// TIA Portal V17 export
// export: Created 2025-03-05T08:01:01.1286192Z, ExportSetting WithDefaults, DisplayName Totally Integrated Automation Portal, DisplayVersion V17 Update 8, DisplayName TIA Portal Openness, DisplayVersion V17 Update 8, DisplayName TIA Portal Version Control Interface, DisplayVersion V17, DisplayName SINAMICS Startdrive Advanced, DisplayVersion V17 SP2, DisplayName SINAMICS Startdrive G110M, G120, G120C, G120D, G120P, G115D, DisplayVersion V17 SP2, DisplayName SINAMICS Startdrive G130, G150, S120, S150, SINAMICS MV, S210, DisplayVersion V17 SP2, DisplayName STEP 7 Professional, DisplayVersion V17 Update 8, DisplayName SINUMERIK ONE STEP 7 Toolbox, DisplayVersion V17 Update 12, DisplayName SINUMERIK 840D sl STEP 7 Toolbox, DisplayVersion V17 Update 12, DisplayName STEP 7 Safety, DisplayVersion V17 Update 6, DisplayName WinCC Advanced, DisplayVersion V17 Update 8
DATA_BLOCK "LTLP_HMIProInterfaceData"   // DB501
{ S7_Optimized_Access := 'FALSE'; DB_Accessible_From_OPC_UA := 'FALSE' }
AUTHOR : TL_TYP6
FAMILY : TL
NAME : UDT_HMI
VERSION : 4.0
// stored: AutoNumber false, DBAccessibleFromOPCUA false, DBAccessibleFromWebserver true, InstanceOfName LTLP_typeHmiProInterface, InstanceOfType UDT, IsOnlyStoredInLoadMemory false, IsWriteProtectedInAS false
"LTLP_typeHmiProInterface"
   // VAR RETAIN
   //    nameStation : Array[1..8] of Char;
   //    noDBWorkpieceCount32 : Int;
   //    startDBWorkpieceCount32 : Int;
   //    cntWorkpiecetypes : Int;
   //    currentProtectLevel : Byte;
   //    eksIdent1 : Byte;
   //    eksIdent2 : Byte;
   //    eksIdent3 : Byte;
   //    eksIdent4 : Byte;
   //    eksIdent5 : Byte;
   //    eksIdent6 : Byte;
   //    eksIdent7 : Byte;
   //    eksOperatorIdentification : Byte;
   //    eksIdent8 : Byte;
   //    res24 : Array[24..31] of Byte;
   //    eksPLCSwitchover : Byte;
   //    res33 : Array[34..47] of Byte;
   //    byte480 : Byte;
   //    netIndex : Byte;
   //    resWinBDE : Array[50..53] of Byte;
   //    selWorkpiecetypePreselect : Word;
   //    selWorkpieceCountReset : Word;
   //    resetTotalCounter : Bool;
   //    resetDailyCounter : Bool;
   //    resetShiftCounter : Bool;
   //    res60 : Array[60..67] of Byte;
   //    codeWorkpiece : Word;
   //    selectProtectionDoors : Bool;
   //    reserve70p1 : Bool;
   //    reserve70p2 : Bool;
   //    reserve70p3 : Bool;
   //    reserve70p4 : Bool;
   //    reserve70p5 : Bool;
   //    reserve70p6 : Bool;
   //    reserve70p7 : Bool;
   //    reserve70p8 : Bool;
   //    reserve70p9 : Bool;
   //    reserve70p10 : Bool;
   //    reserve70p11 : Bool;
   //    reserve70p12 : Bool;
   //    reserve70p13 : Bool;
   //    reserve70p14 : Bool;
   //    reserve70p15 : Bool;
   //    noFunctionKeySubscreen : Word;
   //    selToolGroup : Byte;
   //    toolExtendingServiceLife : Bool;
   //    toolReactivating : Bool;
   //    toolDisable : Bool;
   //    res753 : Bool;
   //    res754 : Bool;
   //    res755 : Bool;
   //    res756 : Bool;
   //    res757 : Bool;
   //    controlPanelOk : Bool;
   //    pAutomaticMode : Bool;
   //    pSingleMode : Bool;
   //    pSingleStepMode : Bool;
   //    pSetupMode : Bool;
   //    pAllUnitsBack : Bool;
   //    pMachineOff : Bool;
   //    p6 : Bool;
   //    p7 : Bool;
   //    pPlus : Bool;
   //    pMinus : Bool;
   //    pEmergencyStop : Bool;
   //    pFaultWillBeCorrected : Bool;
   //    pStart : Bool;
   //    pBasicPosition : Bool;
   //    pMachineOn : Bool;
   //    pGroupAcknowledge : Bool;
   //    pReset : Bool;
   //    pLamptest : Bool;
   //    pRunmode_sweep : Bool;
   //    pMessageAcknowledge : Bool;
   //    pPartCounterReset : Bool;
   //    noFunctionLow : Byte;
   //    noFunctionHigh : Byte;
   //    pStopAfterEndOfCycle : Bool;
   //    pImmediateStop : Bool;
   //    pBridgeEnablingButton : Bool;
   //    pConnectEnablingButton : Bool;
   //    pLockReleaseProtectDoors : Bool;
   //    pMediaOn : Bool;
   //    pMediaOff : Bool;
   //    noSoftKey : Byte;
   //    noFunctionKey : Byte;
   //    noScreenId : Word;
   //    automaticModeCompleteMachine : Bool;
   //    automaticMode : Bool;
   //    singleMode : Bool;
   //    singleStepMode : Bool;
   //    setupMode : Bool;
   //    completionReport : Bool;
   //    gotoBasicPosition : Bool;
   //    reachedBasicPosition : Bool;
   //    startJog : Bool;
   //    immediateStop : Bool;
   //    selStopAfterEndOfCycle : Bool;
   //    reachedStopAfterEndOfCycle : Bool;
   //    motionPlus : Bool;
   //    motionMinus : Bool;
   //    machineUnitOn : Bool;
   //    machineUnitOff : Bool;
   //    allUnitsBack : Bool;
   //    accessAuthorized : Bool;
   //    generalFault : Bool;
   //    executionFault : Bool;
   //    warningOperationalMessage : Bool;
   //    completeMachineFault : Bool;
   //    completeMachineBasicPosition : Bool;
   //    completeMachineCompletReport { ExternalWritable := 'False'} : Bool;
   //    faPartMachining : Bool;
   //    load : Bool;
   //    withoutMachining : Bool;
   //    toolGroupAckOrEnable : Bool;
   //    readyAutomaticStart : Bool;
   //    res895 : Bool;
   //    res896 : Bool;
   //    res897 : Bool;
   //    cycletypes : Array[1..16] of Bool;
   //    protectiveDoorBridged : Bool;
   //    faultWillBeCorrected : Bool;
   //    BridgeEnablingButton : Bool;
   //    connectEnablingButton : Bool;
   //    groupBitProtectDoorsopen : Bool;
   //    headerSwitchover : Bool;
   //    machineUtilization : Bool;
   //    message : Bool;
   //    logisticsFault : Bool;
   //    globalSupplyOutfeed : Bool;
   //    idleCycles : Bool;
   //    toolChangeAlarm : Bool;
   //    automaticToolChangePosition : Bool;
   //    updateRequest : Bool;
   //    toolChangeWarning : Bool;
   //    learnToolChangeSystemActive : Bool;
   //    headerText1 : Bool;
   //    headerText2 : Bool;
   //    headerText3 : Bool;
   //    headerText4 : Bool;
   //    headerText5 : Bool;
   //    headerText6 : Bool;
   //    headerText7 : Bool;
   //    headerText8 : Bool;
   //    automaticStart : Bool;
   //    manualMode : Bool;
   //    transportPosition : Bool;
   //    handHeldUnit : Bool;
   //    mediaOn : Bool;
   //    mediaOff : Bool;
   //    lockReleaseProtectDoors : Bool;
   //    lockingScreenSwitchover : Bool;
   //    exitIsOccupied : Bool;
   //    noPartAtInfeed : Bool;
   //    noFeedParts : Bool;
   //    changeLanguage : Bool;
   //    TriggBitReadPartId : Bool;
   //    cycleBitShiftRegPartId : Bool;
   //    disableDataAvailable : Bool;
   //    upsResponded : Bool;
   //    pageId : Byte;
   //    shiftNumber : Byte;
   //    partsPerCycle : Byte;
   //    taskTriggFeedbackRecipe : Byte;
   //    noControlRecipe : Byte;
   //    nameScreenRecipe : Array[1..27] of Char;
   //    movement1EndPosLeft : Bool;   // Setup screen: left end position of movement reached
   //    movement1EndPosRight : Bool;   // Setup screen: right end position of movement reached
   //    movement2EndPosLeft : Bool;   // Setup screen: left end position of movement reached
   //    movement2EndPosRight : Bool;   // Setup screen: right end position of movement reached
   //    movement3EndPosLeft : Bool;   // Setup screen: left end position of movement reached
   //    movement3EndPosRight : Bool;   // Setup screen: right end position of movement reached
   //    movement4EndPosLeft : Bool;   // Setup screen: left end position of movement reached
   //    movement4EndPosRight : Bool;   // Setup screen: right end position of movement reached
   //    movement5EndPosLeft : Bool;   // Setup screen: left end position of movement reached
   //    movement5EndPosRight : Bool;   // Setup screen: right end position of movement reached
   //    movement6EndPosLeft : Bool;   // Setup screen: left end position of movement reached
   //    movement6EndPosRight : Bool;   // Setup screen: right end position of movement reached
   //    movement7EndPosLeft : Bool;   // Setup screen: left end position of movement reached
   //    movement7EndPosRight : Bool;   // Setup screen: right end position of movement reached
   //    movement8EndPosLeft : Bool;   // Setup screen: left end position of movement reached
   //    movement8EndPosRight : Bool;   // Setup screen: right end position of movement reached
   //    movement9EndPosLeft : Bool;   // Setup screen: left end position of movement reached
   //    movement9EndPosRight : Bool;   // Setup screen: right end position of movement reached
   //    movement10EndPosLeft : Bool;   // Setup screen: left end position of movement reached
   //    movement10EndPosRight : Bool;   // Setup screen: right end position of movement reached
   //    movement11EndPosLeft : Bool;   // Setup screen: left end position of movement reached
   //    movement11EndPosRight : Bool;   // Setup screen: right end position of movement reached
   //    movement12EndPosLeft : Bool;   // Setup screen: left end position of movement reached
   //    movement12EndPosRight : Bool;   // Setup screen: right end position of movement reached
   //    movement13EndPosLeft : Bool;   // Setup screen: left end position of movement reached
   //    movement13EndPosRight : Bool;   // Setup screen: right end position of movement reached
   //    movement14EndPosLeft : Bool;   // Setup screen: left end position of movement reached
   //    movement14EndPosRight : Bool;   // Setup screen: right end position of movement reached
   //    movement15EndPosLeft : Bool;   // Setup screen: left end position of movement reached
   //    movement15EndPosRight : Bool;   // Setup screen: right end position of movement reached
   //    movement16EndPosLeft : Bool;   // Setup screen: left end position of movement reached
   //    movement16EndPosRight : Bool;   // Setup screen: right end position of movement reached
   //    movement17EndPosLeft : Bool;   // Setup screen: left end position of movement reached
   //    movement17EndPosRight : Bool;   // Setup screen: right end position of movement reached
   //    movement18EndPosLeft : Bool;   // Setup screen: left end position of movement reached
   //    movement18EndPosRight : Bool;   // Setup screen: right end position of movement reached
   //    movement19EndPosLeft : Bool;   // Setup screen: left end position of movement reached
   //    movement19EndPosRight : Bool;   // Setup screen: right end position of movement reached
   //    movement20EndPosLeft : Bool;   // Setup screen: left end position of movement reached
   //    movement20EndPosRight : Bool;   // Setup screen: right end position of movement reached
   //    movement21EndPosLeft : Bool;   // Setup screen: left end position of movement reached
   //    movement21EndPosRight : Bool;   // Setup screen: right end position of movement reached
   //    movement22EndPosLeft : Bool;   // Setup screen: left end position of movement reached
   //    movement22EndPosRight : Bool;   // Setup screen: right end position of movement reached
   //    movement23EndPosLeft : Bool;   // Setup screen: left end position of movement reached
   //    movement23EndPosRight : Bool;   // Setup screen: right end position of movement reached
   //    movement24EndPosLeft : Bool;   // Setup screen: left end position of movement reached
   //    movement24EndPosRight : Bool;   // Setup screen: right end position of movement reached
   //    movement25EndPosLeft : Bool;   // Setup screen: left end position of movement reached
   //    movement25EndPosRight : Bool;   // Setup screen: right end position of movement reached
   //    movement26EndPosLeft : Bool;   // Setup screen: left end position of movement reached
   //    movement26EndPosRight : Bool;   // Setup screen: right end position of movement reached
   //    movement27EndPosLeft : Bool;   // Setup screen: left end position of movement reached
   //    movement27EndPosRight : Bool;   // Setup screen: right end position of movement reached
   //    movement28EndPosLeft : Bool;   // Setup screen: left end position of movement reached
   //    movement28EndPosRight : Bool;   // Setup screen: right end position of movement reached
   //    movement29EndPosLeft : Bool;   // Setup screen: left end position of movement reached
   //    movement29EndPosRight : Bool;   // Setup screen: right end position of movement reached
   //    movement30EndPosLeft : Bool;   // Setup screen: left end position of movement reached
   //    movement30EndPosRight : Bool;   // Setup screen: right end position of movement reached
   //    movement31EndPosLeft : Bool;   // Setup screen: left end position of movement reached
   //    movement31EndPosRight : Bool;   // Setup screen: right end position of movement reached
   //    movement32EndPosLeft : Bool;   // Setup screen: left end position of movement reached
   //    movement32EndPosRight : Bool;   // Setup screen: right end position of movement reached
   //    movement33EndPosLeft : Bool;   // Setup screen: left end position of movement reached
   //    movement33EndPosRight : Bool;   // Setup screen: right end position of movement reached
   //    movement34EndPosLeft : Bool;   // Setup screen: left end position of movement reached
   //    movement34EndPosRight : Bool;   // Setup screen: right end position of movement reached
   //    movement35EndPosLeft : Bool;   // Setup screen: left end position of movement reached
   //    movement35EndPosRight : Bool;   // Setup screen: right end position of movement reached
   //    movement36EndPosLeft : Bool;   // Setup screen: left end position of movement reached
   //    movement36EndPosRight : Bool;   // Setup screen: right end position of movement reached
   //    movement37EndPosLeft : Bool;   // Setup screen: left end position of movement reached
   //    movement37EndPosRight : Bool;   // Setup screen: right end position of movement reached
   //    movement38EndPosLeft : Bool;   // Setup screen: left end position of movement reached
   //    movement38EndPosRight : Bool;   // Setup screen: right end position of movement reached
   //    movement39EndPosLeft : Bool;   // Setup screen: left end position of movement reached
   //    movement39EndPosRight : Bool;   // Setup screen: right end position of movement reached
   //    movement40EndPosLeft : Bool;   // Setup screen: left end position of movement reached
   //    movement40EndPosRight : Bool;   // Setup screen: right end position of movement reached
   //    movement41EndPosLeft : Bool;   // Setup screen: left end position of movement reached
   //    movement41EndPosRight : Bool;   // Setup screen: right end position of movement reached
   //    movement42EndPosLeft : Bool;   // Setup screen: left end position of movement reached
   //    movement42EndPosRight : Bool;   // Setup screen: right end position of movement reached
   //    movement43EndPosLeft : Bool;   // Setup screen: left end position of movement reached
   //    movement43EndPosRight : Bool;   // Setup screen: right end position of movement reached
   //    movement44EndPosLeft : Bool;   // Setup screen: left end position of movement reached
   //    movement44EndPosRight : Bool;   // Setup screen: right end position of movement reached
   //    movement45EndPosLeft : Bool;   // Setup screen: left end position of movement reached
   //    movement45EndPosRight : Bool;   // Setup screen: right end position of movement reached
   //    movement46EndPosLeft : Bool;   // Setup screen: left end position of movement reached
   //    movement46EndPosRight : Bool;   // Setup screen: right end position of movement reached
   //    movement47EndPosLeft : Bool;   // Setup screen: left end position of movement reached
   //    movement47EndPosRight : Bool;   // Setup screen: right end position of movement reached
   //    movement48EndPosLeft : Bool;   // Setup screen: left end position of movement reached
   //    movement48EndPosRight : Bool;   // Setup screen: right end position of movement reached
   //    movement49EndPosLeft : Bool;   // Setup screen: left end position of movement reached
   //    movement49EndPosRight : Bool;   // Setup screen: right end position of movement reached
   //    movement50EndPosLeft : Bool;   // Setup screen: left end position of movement reached
   //    movement50EndPosRight : Bool;   // Setup screen: right end position of movement reached
   //    movement51EndPosLeft : Bool;   // Setup screen: left end position of movement reached
   //    movement51EndPosRight : Bool;   // Setup screen: right end position of movement reached
   //    movement52EndPosLeft : Bool;   // Setup screen: left end position of movement reached
   //    movement52EndPosRight : Bool;   // Setup screen: right end position of movement reached
   //    movement53EndPosLeft : Bool;   // Setup screen: left end position of movement reached
   //    movement53EndPosRight : Bool;   // Setup screen: right end position of movement reached
   //    movement54EndPosLeft : Bool;   // Setup screen: left end position of movement reached
   //    movement54EndPosRight : Bool;   // Setup screen: right end position of movement reached
   //    movement55EndPosLeft : Bool;   // Setup screen: left end position of movement reached
   //    movement55EndPosRight : Bool;   // Setup screen: right end position of movement reached
   //    movement56EndPosLeft : Bool;   // Setup screen: left end position of movement reached
   //    movement56EndPosRight : Bool;   // Setup screen: right end position of movement reached
   //    movement57EndPosLeft : Bool;   // Setup screen: left end position of movement reached
   //    movement57EndPosRight : Bool;   // Setup screen: right end position of movement reached
   //    movement58EndPosLeft : Bool;   // Setup screen: left end position of movement reached
   //    movement58EndPosRight : Bool;   // Setup screen: right end position of movement reached
   //    movement59EndPosLeft : Bool;   // Setup screen: left end position of movement reached
   //    movement59EndPosRight : Bool;   // Setup screen: right end position of movement reached
   //    movement60EndPosLeft : Bool;   // Setup screen: left end position of movement reached
   //    movement60EndPosRight : Bool;   // Setup screen: right end position of movement reached
   //    movement61EndPosLeft : Bool;   // Setup screen: left end position of movement reached
   //    movement61EndPosRight : Bool;   // Setup screen: right end position of movement reached
   //    movement62EndPosLeft : Bool;   // Setup screen: left end position of movement reached
   //    movement62EndPosRight : Bool;   // Setup screen: right end position of movement reached
   //    movement63EndPosLeft : Bool;   // Setup screen: left end position of movement reached
   //    movement63EndPosRight : Bool;   // Setup screen: right end position of movement reached
   //    movement64EndPosLeft : Bool;   // Setup screen: left end position of movement reached
   //    movement64EndPosRight : Bool;   // Setup screen: right end position of movement reached
   //    movement65EndPosLeft : Bool;   // Setup screen: left end position of movement reached
   //    movement65EndPosRight : Bool;   // Setup screen: right end position of movement reached
   //    movement66EndPosLeft : Bool;   // Setup screen: left end position of movement reached
   //    movement66EndPosRight : Bool;   // Setup screen: right end position of movement reached
   //    movement67EndPosLeft : Bool;   // Setup screen: left end position of movement reached
   //    movement67EndPosRight : Bool;   // Setup screen: right end position of movement reached
   //    movement68EndPosLeft : Bool;   // Setup screen: left end position of movement reached
   //    movement68EndPosRight : Bool;   // Setup screen: right end position of movement reached
   //    movement69EndPosLeft : Bool;   // Setup screen: left end position of movement reached
   //    movement69EndPosRight : Bool;   // Setup screen: right end position of movement reached
   //    movement70EndPosLeft : Bool;   // Setup screen: left end position of movement reached
   //    movement70EndPosRight : Bool;   // Setup screen: right end position of movement reached
   //    movement71EndPosLeft : Bool;   // Setup screen: left end position of movement reached
   //    movement71EndPosRight : Bool;   // Setup screen: right end position of movement reached
   //    movement72EndPosLeft : Bool;   // Setup screen: left end position of movement reached
   //    movement72EndPosRight : Bool;   // Setup screen: right end position of movement reached
   //    movement73EndPosLeft : Bool;   // Setup screen: left end position of movement reached
   //    movement73EndPosRight : Bool;   // Setup screen: right end position of movement reached
   //    movement74EndPosLeft : Bool;   // Setup screen: left end position of movement reached
   //    movement74EndPosRight : Bool;   // Setup screen: right end position of movement reached
   //    movement75EndPosLeft : Bool;   // Setup screen: left end position of movement reached
   //    movement75EndPosRight : Bool;   // Setup screen: right end position of movement reached
   //    movement76EndPosLeft : Bool;   // Setup screen: left end position of movement reached
   //    movement76EndPosRight : Bool;   // Setup screen: right end position of movement reached
   //    movement77EndPosLeft : Bool;   // Setup screen: left end position of movement reached
   //    movement77EndPosRight : Bool;   // Setup screen: right end position of movement reached
   //    movement78EndPosLeft : Bool;   // Setup screen: left end position of movement reached
   //    movement78EndPosRight : Bool;   // Setup screen: right end position of movement reached
   //    movement79EndPosLeft : Bool;   // Setup screen: left end position of movement reached
   //    movement79EndPosRight : Bool;   // Setup screen: right end position of movement reached
   //    movement80EndPosLeft : Bool;   // Setup screen: left end position of movement reached
   //    movement80EndPosRight : Bool;   // Setup screen: right end position of movement reached
   //    movement81EndPosLeft : Bool;   // Setup screen: left end position of movement reached
   //    movement81EndPosRight : Bool;   // Setup screen: right end position of movement reached
   //    movement82EndPosLeft : Bool;   // Setup screen: left end position of movement reached
   //    movement82EndPosRight : Bool;   // Setup screen: right end position of movement reached
   //    movement83EndPosLeft : Bool;   // Setup screen: left end position of movement reached
   //    movement83EndPosRight : Bool;   // Setup screen: right end position of movement reached
   //    movement84EndPosLeft : Bool;   // Setup screen: left end position of movement reached
   //    movement84EndPosRight : Bool;   // Setup screen: right end position of movement reached
   //    movement85EndPosLeft : Bool;   // Setup screen: left end position of movement reached
   //    movement85EndPosRight : Bool;   // Setup screen: right end position of movement reached
   //    movement86EndPosLeft : Bool;   // Setup screen: left end position of movement reached
   //    movement86EndPosRight : Bool;   // Setup screen: right end position of movement reached
   //    movement87EndPosLeft : Bool;   // Setup screen: left end position of movement reached
   //    movement87EndPosRight : Bool;   // Setup screen: right end position of movement reached
   //    movement88EndPosLeft : Bool;   // Setup screen: left end position of movement reached
   //    movement88EndPosRight : Bool;   // Setup screen: right end position of movement reached
   //    movement89EndPosLeft : Bool;   // Setup screen: left end position of movement reached
   //    movement89EndPosRight : Bool;   // Setup screen: right end position of movement reached
   //    movement90EndPosLeft : Bool;   // Setup screen: left end position of movement reached
   //    movement90EndPosRight : Bool;   // Setup screen: right end position of movement reached
   //    movement91EndPosLeft : Bool;   // Setup screen: left end position of movement reached
   //    movement91EndPosRight : Bool;   // Setup screen: right end position of movement reached
   //    movement92EndPosLeft : Bool;   // Setup screen: left end position of movement reached
   //    movement92EndPosRight : Bool;   // Setup screen: right end position of movement reached
   //    movement93EndPosLeft : Bool;   // Setup screen: left end position of movement reached
   //    movement93EndPosRight : Bool;   // Setup screen: right end position of movement reached
   //    movement94EndPosLeft : Bool;   // Setup screen: left end position of movement reached
   //    movement94EndPosRight : Bool;   // Setup screen: right end position of movement reached
   //    movement95EndPosLeft : Bool;   // Setup screen: left end position of movement reached
   //    movement95EndPosRight : Bool;   // Setup screen: right end position of movement reached
   //    movement96EndPosLeft : Bool;   // Setup screen: left end position of movement reached
   //    movement96EndPosRight : Bool;   // Setup screen: right end position of movement reached
   //    movement97EndPosLeft : Bool;   // Setup screen: left end position of movement reached
   //    movement97EndPosRight : Bool;   // Setup screen: right end position of movement reached
   //    movement98EndPosLeft : Bool;   // Setup screen: left end position of movement reached
   //    movement98EndPosRight : Bool;   // Setup screen: right end position of movement reached
   //    movement99EndPosLeft : Bool;   // Setup screen: left end position of movement reached
   //    movement99EndPosRight : Bool;   // Setup screen: right end position of movement reached
   //    movement100EndPosLeft : Bool;   // Setup screen: left end position of movement reached
   //    movement100EndPosRight : Bool;   // Setup screen: right end position of movement reached
   //    movement101EndPosLeft : Bool;   // Setup screen: left end position of movement reached
   //    movement101EndPosRight : Bool;   // Setup screen: right end position of movement reached
   //    movement102EndPosLeft : Bool;   // Setup screen: left end position of movement reached
   //    movement102EndPosRight : Bool;   // Setup screen: right end position of movement reached
   //    movement103EndPosLeft : Bool;   // Setup screen: left end position of movement reached
   //    movement103EndPosRight : Bool;   // Setup screen: right end position of movement reached
   //    movement104EndPosLeft : Bool;   // Setup screen: left end position of movement reached
   //    movement104EndPosRight : Bool;   // Setup screen: right end position of movement reached
   //    movement105EndPosLeft : Bool;   // Setup screen: left end position of movement reached
   //    movement105EndPosRight : Bool;   // Setup screen: right end position of movement reached
   //    movement106EndPosLeft : Bool;   // Setup screen: left end position of movement reached
   //    movement106EndPosRight : Bool;   // Setup screen: right end position of movement reached
   //    movement107EndPosLeft : Bool;   // Setup screen: left end position of movement reached
   //    movement107EndPosRight : Bool;   // Setup screen: right end position of movement reached
   //    movement108EndPosLeft : Bool;   // Setup screen: left end position of movement reached
   //    movement108EndPosRight : Bool;   // Setup screen: right end position of movement reached
   //    movement109EndPosLeft : Bool;   // Setup screen: left end position of movement reached
   //    movement109EndPosRight : Bool;   // Setup screen: right end position of movement reached
   //    movement110EndPosLeft : Bool;   // Setup screen: left end position of movement reached
   //    movement110EndPosRight : Bool;   // Setup screen: right end position of movement reached
   //    movement111EndPosLeft : Bool;   // Setup screen: left end position of movement reached
   //    movement111EndPosRight : Bool;   // Setup screen: right end position of movement reached
   //    movement112EndPosLeft : Bool;   // Setup screen: left end position of movement reached
   //    movement112EndPosRight : Bool;   // Setup screen: right end position of movement reached
   //    movement113EndPosLeft : Bool;   // Setup screen: left end position of movement reached
   //    movement113EndPosRight : Bool;   // Setup screen: right end position of movement reached
   //    movement114EndPosLeft : Bool;   // Setup screen: left end position of movement reached
   //    movement114EndPosRight : Bool;   // Setup screen: right end position of movement reached
   //    movement115EndPosLeft : Bool;   // Setup screen: left end position of movement reached
   //    movement115EndPosRight : Bool;   // Setup screen: right end position of movement reached
   //    movement116EndPosLeft : Bool;   // Setup screen: left end position of movement reached
   //    movement116EndPosRight : Bool;   // Setup screen: right end position of movement reached
   //    movement117EndPosLeft : Bool;   // Setup screen: left end position of movement reached
   //    movement117EndPosRight : Bool;   // Setup screen: right end position of movement reached
   //    movement118EndPosLeft : Bool;   // Setup screen: left end position of movement reached
   //    movement118EndPosRight : Bool;   // Setup screen: right end position of movement reached
   //    movement119EndPosLeft : Bool;   // Setup screen: left end position of movement reached
   //    movement119EndPosRight : Bool;   // Setup screen: right end position of movement reached
   //    movement120EndPosLeft : Bool;   // Setup screen: left end position of movement reached
   //    movement120EndPosRight : Bool;   // Setup screen: right end position of movement reached
   //    movement121EndPosLeft : Bool;   // Setup screen: left end position of movement reached
   //    movement121EndPosRight : Bool;   // Setup screen: right end position of movement reached
   //    movement122EndPosLeft : Bool;   // Setup screen: left end position of movement reached
   //    movement122EndPosRight : Bool;   // Setup screen: right end position of movement reached
   //    movement123EndPosLeft : Bool;   // Setup screen: left end position of movement reached
   //    movement123EndPosRight : Bool;   // Setup screen: right end position of movement reached
   //    movement124EndPosLeft : Bool;   // Setup screen: left end position of movement reached
   //    movement124EndPosRight : Bool;   // Setup screen: right end position of movement reached
   //    movement125EndPosLeft : Bool;   // Setup screen: left end position of movement reached
   //    movement125EndPosRight : Bool;   // Setup screen: right end position of movement reached
   //    movement126EndPosLeft : Bool;   // Setup screen: left end position of movement reached
   //    movement126EndPosRight : Bool;   // Setup screen: right end position of movement reached
   //    movement127EndPosLeft : Bool;   // Setup screen: left end position of movement reached
   //    movement127EndPosRight : Bool;   // Setup screen: right end position of movement reached
   //    movement128EndPosLeft : Bool;   // Setup screen: left end position of movement reached
   //    movement128EndPosRight : Bool;   // Setup screen: right end position of movement reached
   //    movement129EndPosLeft : Bool;   // Setup screen: left end position of movement reached
   //    movement129EndPosRight : Bool;   // Setup screen: right end position of movement reached
   //    movement130EndPosLeft : Bool;   // Setup screen: left end position of movement reached
   //    movement130EndPosRight : Bool;   // Setup screen: right end position of movement reached
   //    movement131EndPosLeft : Bool;   // Setup screen: left end position of movement reached
   //    movement131EndPosRight : Bool;   // Setup screen: right end position of movement reached
   //    movement132EndPosLeft : Bool;   // Setup screen: left end position of movement reached
   //    movement132EndPosRight : Bool;   // Setup screen: right end position of movement reached
   //    movement133EndPosLeft : Bool;   // Setup screen: left end position of movement reached
   //    movement133EndPosRight : Bool;   // Setup screen: right end position of movement reached
   //    movement134EndPosLeft : Bool;   // Setup screen: left end position of movement reached
   //    movement134EndPosRight : Bool;   // Setup screen: right end position of movement reached
   //    movement135EndPosLeft : Bool;   // Setup screen: left end position of movement reached
   //    movement135EndPosRight : Bool;   // Setup screen: right end position of movement reached
   //    movement136EndPosLeft : Bool;   // Setup screen: left end position of movement reached
   //    movement136EndPosRight : Bool;   // Setup screen: right end position of movement reached
   //    movement137EndPosLeft : Bool;   // Setup screen: left end position of movement reached
   //    movement137EndPosRight : Bool;   // Setup screen: right end position of movement reached
   //    movement138EndPosLeft : Bool;   // Setup screen: left end position of movement reached
   //    movement138EndPosRight : Bool;   // Setup screen: right end position of movement reached
   //    movement139EndPosLeft : Bool;   // Setup screen: left end position of movement reached
   //    movement139EndPosRight : Bool;   // Setup screen: right end position of movement reached
   //    movement140EndPosLeft : Bool;   // Setup screen: left end position of movement reached
   //    movement140EndPosRight : Bool;   // Setup screen: right end position of movement reached
   //    movement141EndPosLeft : Bool;   // Setup screen: left end position of movement reached
   //    movement141EndPosRight : Bool;   // Setup screen: right end position of movement reached
   //    movement142EndPosLeft : Bool;   // Setup screen: left end position of movement reached
   //    movement142EndPosRight : Bool;   // Setup screen: right end position of movement reached
   //    movement143EndPosLeft : Bool;   // Setup screen: left end position of movement reached
   //    movement143EndPosRight : Bool;   // Setup screen: right end position of movement reached
   //    movement144EndPosLeft : Bool;   // Setup screen: left end position of movement reached
   //    movement144EndPosRight : Bool;   // Setup screen: right end position of movement reached
   //    movement145EndPosLeft : Bool;   // Setup screen: left end position of movement reached
   //    movement145EndPosRight : Bool;   // Setup screen: right end position of movement reached
   //    movement146EndPosLeft : Bool;   // Setup screen: left end position of movement reached
   //    movement146EndPosRight : Bool;   // Setup screen: right end position of movement reached
   //    movement147EndPosLeft : Bool;   // Setup screen: left end position of movement reached
   //    movement147EndPosRight : Bool;   // Setup screen: right end position of movement reached
   //    movement148EndPosLeft : Bool;   // Setup screen: left end position of movement reached
   //    movement148EndPosRight : Bool;   // Setup screen: right end position of movement reached
   //    movement149EndPosLeft : Bool;   // Setup screen: left end position of movement reached
   //    movement149EndPosRight : Bool;   // Setup screen: right end position of movement reached
   //    movement150EndPosLeft : Bool;   // Setup screen: left end position of movement reached
   //    movement150EndPosRight : Bool;   // Setup screen: right end position of movement reached
   //    movement151EndPosLeft : Bool;   // Setup screen: left end position of movement reached
   //    movement151EndPosRight : Bool;   // Setup screen: right end position of movement reached
   //    movement152EndPosLeft : Bool;   // Setup screen: left end position of movement reached
   //    movement152EndPosRight : Bool;   // Setup screen: right end position of movement reached
   //    movement153EndPosLeft : Bool;   // Setup screen: left end position of movement reached
   //    movement153EndPosRight : Bool;   // Setup screen: right end position of movement reached
   //    movement154EndPosLeft : Bool;   // Setup screen: left end position of movement reached
   //    movement154EndPosRight : Bool;   // Setup screen: right end position of movement reached
   //    movement155EndPosLeft : Bool;   // Setup screen: left end position of movement reached
   //    movement155EndPosRight : Bool;   // Setup screen: right end position of movement reached
   //    movement156EndPosLeft : Bool;   // Setup screen: left end position of movement reached
   //    movement156EndPosRight : Bool;   // Setup screen: right end position of movement reached
   //    movement157EndPosLeft : Bool;   // Setup screen: left end position of movement reached
   //    movement157EndPosRight : Bool;   // Setup screen: right end position of movement reached
   //    movement158EndPosLeft : Bool;   // Setup screen: left end position of movement reached
   //    movement158EndPosRight : Bool;   // Setup screen: right end position of movement reached
   //    movement159EndPosLeft : Bool;   // Setup screen: left end position of movement reached
   //    movement159EndPosRight : Bool;   // Setup screen: right end position of movement reached
   //    movement160EndPosLeft : Bool;   // Setup screen: left end position of movement reached
   //    movement160EndPosRight : Bool;   // Setup screen: right end position of movement reached
   //    movement161EndPosLeft : Bool;   // Setup screen: left end position of movement reached
   //    movement161EndPosRight : Bool;   // Setup screen: right end position of movement reached
   //    movement162EndPosLeft : Bool;   // Setup screen: left end position of movement reached
   //    movement162EndPosRight : Bool;   // Setup screen: right end position of movement reached
   //    movement163EndPosLeft : Bool;   // Setup screen: left end position of movement reached
   //    movement163EndPosRight : Bool;   // Setup screen: right end position of movement reached
   //    movement164EndPosLeft : Bool;   // Setup screen: left end position of movement reached
   //    movement164EndPosRight : Bool;   // Setup screen: right end position of movement reached
   //    movement165EndPosLeft : Bool;   // Setup screen: left end position of movement reached
   //    movement165EndPosRight : Bool;   // Setup screen: right end position of movement reached
   //    movement166EndPosLeft : Bool;   // Setup screen: left end position of movement reached
   //    movement166EndPosRight : Bool;   // Setup screen: right end position of movement reached
   //    movement167EndPosLeft : Bool;   // Setup screen: left end position of movement reached
   //    movement167EndPosRight : Bool;   // Setup screen: right end position of movement reached
   //    movement168EndPosLeft : Bool;   // Setup screen: left end position of movement reached
   //    movement168EndPosRight : Bool;   // Setup screen: right end position of movement reached
   //    movement169EndPosLeft : Bool;   // Setup screen: left end position of movement reached
   //    movement169EndPosRight : Bool;   // Setup screen: right end position of movement reached
   //    movement170EndPosLeft : Bool;   // Setup screen: left end position of movement reached
   //    movement170EndPosRight : Bool;   // Setup screen: right end position of movement reached
   //    movement171EndPosLeft : Bool;   // Setup screen: left end position of movement reached
   //    movement171EndPosRight : Bool;   // Setup screen: right end position of movement reached
   //    movement172EndPosLeft : Bool;   // Setup screen: left end position of movement reached
   //    movement172EndPosRight : Bool;   // Setup screen: right end position of movement reached
   //    movement173EndPosLeft : Bool;   // Setup screen: left end position of movement reached
   //    movement173EndPosRight : Bool;   // Setup screen: right end position of movement reached
   //    movement174EndPosLeft : Bool;   // Setup screen: left end position of movement reached
   //    movement174EndPosRight : Bool;   // Setup screen: right end position of movement reached
   //    movement175EndPosLeft : Bool;   // Setup screen: left end position of movement reached
   //    movement175EndPosRight : Bool;   // Setup screen: right end position of movement reached
   //    movement176EndPosLeft : Bool;   // Setup screen: left end position of movement reached
   //    movement176EndPosRight : Bool;   // Setup screen: right end position of movement reached
   //    movement177EndPosLeft : Bool;   // Setup screen: left end position of movement reached
   //    movement177EndPosRight : Bool;   // Setup screen: right end position of movement reached
   //    movement178EndPosLeft : Bool;   // Setup screen: left end position of movement reached
   //    movement178EndPosRight : Bool;   // Setup screen: right end position of movement reached
   //    movement179EndPosLeft : Bool;   // Setup screen: left end position of movement reached
   //    movement179EndPosRight : Bool;   // Setup screen: right end position of movement reached
   //    movement180EndPosLeft : Bool;   // Setup screen: left end position of movement reached
   //    movement180EndPosRight : Bool;   // Setup screen: right end position of movement reached
   //    movement181EndPosLeft : Bool;   // Setup screen: left end position of movement reached
   //    movement181EndPosRight : Bool;   // Setup screen: right end position of movement reached
   //    movement182EndPosLeft : Bool;   // Setup screen: left end position of movement reached
   //    movement182EndPosRight : Bool;   // Setup screen: right end position of movement reached
   //    movement183EndPosLeft : Bool;   // Setup screen: left end position of movement reached
   //    movement183EndPosRight : Bool;   // Setup screen: right end position of movement reached
   //    movement184EndPosLeft : Bool;   // Setup screen: left end position of movement reached
   //    movement184EndPosRight : Bool;   // Setup screen: right end position of movement reached
   //    movement185EndPosLeft : Bool;   // Setup screen: left end position of movement reached
   //    movement185EndPosRight : Bool;   // Setup screen: right end position of movement reached
   //    movement186EndPosLeft : Bool;   // Setup screen: left end position of movement reached
   //    movement186EndPosRight : Bool;   // Setup screen: right end position of movement reached
   //    movement187EndPosLeft : Bool;   // Setup screen: left end position of movement reached
   //    movement187EndPosRight : Bool;   // Setup screen: right end position of movement reached
   //    movement188EndPosLeft : Bool;   // Setup screen: left end position of movement reached
   //    movement188EndPosRight : Bool;   // Setup screen: right end position of movement reached
   //    movement189EndPosLeft : Bool;   // Setup screen: left end position of movement reached
   //    movement189EndPosRight : Bool;   // Setup screen: right end position of movement reached
   //    movement190EndPosLeft : Bool;   // Setup screen: left end position of movement reached
   //    movement190EndPosRight : Bool;   // Setup screen: right end position of movement reached
   //    movement191EndPosLeft : Bool;   // Setup screen: left end position of movement reached
   //    movement191EndPosRight : Bool;   // Setup screen: right end position of movement reached
   //    movement192EndPosLeft : Bool;   // Setup screen: left end position of movement reached
   //    movement192EndPosRight : Bool;   // Setup screen: right end position of movement reached
   //    movement193EndPosLeft : Bool;   // Setup screen: left end position of movement reached
   //    movement193EndPosRight : Bool;   // Setup screen: right end position of movement reached
   //    movement194EndPosLeft : Bool;   // Setup screen: left end position of movement reached
   //    movement194EndPosRight : Bool;   // Setup screen: right end position of movement reached
   //    movement195EndPosLeft : Bool;   // Setup screen: left end position of movement reached
   //    movement195EndPosRight : Bool;   // Setup screen: right end position of movement reached
   //    movement196EndPosLeft : Bool;   // Setup screen: left end position of movement reached
   //    movement196EndPosRight : Bool;   // Setup screen: right end position of movement reached
   //    movement197EndPosLeft : Bool;   // Setup screen: left end position of movement reached
   //    movement197EndPosRight : Bool;   // Setup screen: right end position of movement reached
   //    movement198EndPosLeft : Bool;   // Setup screen: left end position of movement reached
   //    movement198EndPosRight : Bool;   // Setup screen: right end position of movement reached
   //    movement199EndPosLeft : Bool;   // Setup screen: left end position of movement reached
   //    movement199EndPosRight : Bool;   // Setup screen: right end position of movement reached
   //    movement200EndPosLeft : Bool;   // Setup screen: left end position of movement reached
   //    movement200EndPosRight : Bool;   // Setup screen: right end position of movement reached
   //    movement201EndPosLeft : Bool;   // Setup screen: left end position of movement reached
   //    movement201EndPosRight : Bool;   // Setup screen: right end position of movement reached
   //    movement202EndPosLeft : Bool;   // Setup screen: left end position of movement reached
   //    movement202EndPosRight : Bool;   // Setup screen: right end position of movement reached
   //    movement203EndPosLeft : Bool;   // Setup screen: left end position of movement reached
   //    movement203EndPosRight : Bool;   // Setup screen: right end position of movement reached
   //    movement204EndPosLeft : Bool;   // Setup screen: left end position of movement reached
   //    movement204EndPosRight : Bool;   // Setup screen: right end position of movement reached
   //    movement205EndPosLeft : Bool;   // Setup screen: left end position of movement reached
   //    movement205EndPosRight : Bool;   // Setup screen: right end position of movement reached
   //    movement206EndPosLeft : Bool;   // Setup screen: left end position of movement reached
   //    movement206EndPosRight : Bool;   // Setup screen: right end position of movement reached
   //    movement207EndPosLeft : Bool;   // Setup screen: left end position of movement reached
   //    movement207EndPosRight : Bool;   // Setup screen: right end position of movement reached
   //    movement208EndPosLeft : Bool;   // Setup screen: left end position of movement reached
   //    movement208EndPosRight : Bool;   // Setup screen: right end position of movement reached
   //    movement209EndPosLeft : Bool;   // Setup screen: left end position of movement reached
   //    movement209EndPosRight : Bool;   // Setup screen: right end position of movement reached
   //    movement210EndPosLeft : Bool;   // Setup screen: left end position of movement reached
   //    movement210EndPosRight : Bool;   // Setup screen: right end position of movement reached
   //    movement211EndPosLeft : Bool;   // Setup screen: left end position of movement reached
   //    movement211EndPosRight : Bool;   // Setup screen: right end position of movement reached
   //    movement212EndPosLeft : Bool;   // Setup screen: left end position of movement reached
   //    movement212EndPosRight : Bool;   // Setup screen: right end position of movement reached
   //    movement213EndPosLeft : Bool;   // Setup screen: left end position of movement reached
   //    movement213EndPosRight : Bool;   // Setup screen: right end position of movement reached
   //    movement214EndPosLeft : Bool;   // Setup screen: left end position of movement reached
   //    movement214EndPosRight : Bool;   // Setup screen: right end position of movement reached
   //    movement215EndPosLeft : Bool;   // Setup screen: left end position of movement reached
   //    movement215EndPosRight : Bool;   // Setup screen: right end position of movement reached
   //    movement216EndPosLeft : Bool;   // Setup screen: left end position of movement reached
   //    movement216EndPosRight : Bool;   // Setup screen: right end position of movement reached
   //    movement217EndPosLeft : Bool;   // Setup screen: left end position of movement reached
   //    movement217EndPosRight : Bool;   // Setup screen: right end position of movement reached
   //    movement218EndPosLeft : Bool;   // Setup screen: left end position of movement reached
   //    movement218EndPosRight : Bool;   // Setup screen: right end position of movement reached
   //    movement219EndPosLeft : Bool;   // Setup screen: left end position of movement reached
   //    movement219EndPosRight : Bool;   // Setup screen: right end position of movement reached
   //    movement220EndPosLeft : Bool;   // Setup screen: left end position of movement reached
   //    movement220EndPosRight : Bool;   // Setup screen: right end position of movement reached
   //    movement221EndPosLeft : Bool;   // Setup screen: left end position of movement reached
   //    movement221EndPosRight : Bool;   // Setup screen: right end position of movement reached
   //    movement222EndPosLeft : Bool;   // Setup screen: left end position of movement reached
   //    movement222EndPosRight : Bool;   // Setup screen: right end position of movement reached
   //    movement223EndPosLeft : Bool;   // Setup screen: left end position of movement reached
   //    movement223EndPosRight : Bool;   // Setup screen: right end position of movement reached
   //    movement224EndPosLeft : Bool;   // Setup screen: left end position of movement reached
   //    movement224EndPosRight : Bool;   // Setup screen: right end position of movement reached
   //    movement225EndPosLeft : Bool;   // Setup screen: left end position of movement reached
   //    movement225EndPosRight : Bool;   // Setup screen: right end position of movement reached
   //    movement226EndPosLeft : Bool;   // Setup screen: left end position of movement reached
   //    movement226EndPosRight : Bool;   // Setup screen: right end position of movement reached
   //    movement227EndPosLeft : Bool;   // Setup screen: left end position of movement reached
   //    movement227EndPosRight : Bool;   // Setup screen: right end position of movement reached
   //    movement228EndPosLeft : Bool;   // Setup screen: left end position of movement reached
   //    movement228EndPosRight : Bool;   // Setup screen: right end position of movement reached
   //    movement229EndPosLeft : Bool;   // Setup screen: left end position of movement reached
   //    movement229EndPosRight : Bool;   // Setup screen: right end position of movement reached
   //    movement230EndPosLeft : Bool;   // Setup screen: left end position of movement reached
   //    movement230EndPosRight : Bool;   // Setup screen: right end position of movement reached
   //    movement231EndPosLeft : Bool;   // Setup screen: left end position of movement reached
   //    movement231EndPosRight : Bool;   // Setup screen: right end position of movement reached
   //    movement232EndPosLeft : Bool;   // Setup screen: left end position of movement reached
   //    movement232EndPosRight : Bool;   // Setup screen: right end position of movement reached
   //    movement233EndPosLeft : Bool;   // Setup screen: left end position of movement reached
   //    movement233EndPosRight : Bool;   // Setup screen: right end position of movement reached
   //    movement234EndPosLeft : Bool;   // Setup screen: left end position of movement reached
   //    movement234EndPosRight : Bool;   // Setup screen: right end position of movement reached
   //    movement235EndPosLeft : Bool;   // Setup screen: left end position of movement reached
   //    movement235EndPosRight : Bool;   // Setup screen: right end position of movement reached
   //    movement236EndPosLeft : Bool;   // Setup screen: left end position of movement reached
   //    movement236EndPosRight : Bool;   // Setup screen: right end position of movement reached
   //    movement237EndPosLeft : Bool;   // Setup screen: left end position of movement reached
   //    movement237EndPosRight : Bool;   // Setup screen: right end position of movement reached
   //    movement238EndPosLeft : Bool;   // Setup screen: left end position of movement reached
   //    movement238EndPosRight : Bool;   // Setup screen: right end position of movement reached
   //    movement239EndPosLeft : Bool;   // Setup screen: left end position of movement reached
   //    movement239EndPosRight : Bool;   // Setup screen: right end position of movement reached
   //    movement240EndPosLeft : Bool;   // Setup screen: left end position of movement reached
   //    movement240EndPosRight : Bool;   // Setup screen: right end position of movement reached
   //    movement241EndPosLeft : Bool;   // Setup screen: left end position of movement reached
   //    movement241EndPosRight : Bool;   // Setup screen: right end position of movement reached
   //    movement242EndPosLeft : Bool;   // Setup screen: left end position of movement reached
   //    movement242EndPosRight : Bool;   // Setup screen: right end position of movement reached
   //    movement243EndPosLeft : Bool;   // Setup screen: left end position of movement reached
   //    movement243EndPosRight : Bool;   // Setup screen: right end position of movement reached
   //    movement244EndPosLeft : Bool;   // Setup screen: left end position of movement reached
   //    movement244EndPosRight : Bool;   // Setup screen: right end position of movement reached
   //    movement245EndPosLeft : Bool;   // Setup screen: left end position of movement reached
   //    movement245EndPosRight : Bool;   // Setup screen: right end position of movement reached
   //    movement246EndPosLeft : Bool;   // Setup screen: left end position of movement reached
   //    movement246EndPosRight : Bool;   // Setup screen: right end position of movement reached
   //    movement247EndPosLeft : Bool;   // Setup screen: left end position of movement reached
   //    movement247EndPosRight : Bool;   // Setup screen: right end position of movement reached
   //    movement248EndPosLeft : Bool;   // Setup screen: left end position of movement reached
   //    movement248EndPosRight : Bool;   // Setup screen: right end position of movement reached
   //    movement249EndPosLeft : Bool;   // Setup screen: left end position of movement reached
   //    movement249EndPosRight : Bool;   // Setup screen: right end position of movement reached
   //    movement250EndPosLeft : Bool;   // Setup screen: left end position of movement reached
   //    movement250EndPosRight : Bool;   // Setup screen: right end position of movement reached
   //    movement251EndPosLeft : Bool;   // Setup screen: left end position of movement reached
   //    movement251EndPosRight : Bool;   // Setup screen: right end position of movement reached
   //    movement252EndPosLeft : Bool;   // Setup screen: left end position of movement reached
   //    movement252EndPosRight : Bool;   // Setup screen: right end position of movement reached
   //    movement253EndPosLeft : Bool;   // Setup screen: left end position of movement reached
   //    movement253EndPosRight : Bool;   // Setup screen: right end position of movement reached
   //    movement254EndPosLeft : Bool;   // Setup screen: left end position of movement reached
   //    movement254EndPosRight : Bool;   // Setup screen: right end position of movement reached
   //    movement255EndPosLeft : Bool;   // Setup screen: left end position of movement reached
   //    movement255EndPosRight : Bool;   // Setup screen: right end position of movement reached
   //    movement256EndPosLeft : Bool;   // Setup screen: left end position of movement reached
   //    movement256EndPosRight : Bool;   // Setup screen: right end position of movement reached
   //    res194 : Array[1..16] of Bool;
   //    res196 : Word;
   //    movement1ExecutabilityLeft : Bool;   // Setup screen: executability of movement left
   //    movement1ExecutabilityRight : Bool;   // Setup screen: executability of movement right
   //    movement2ExecutabilityLeft : Bool;   // Setup screen: executability of movement left
   //    movement2ExecutabilityRight : Bool;   // Setup screen: executability of movement right
   //    movement3ExecutabilityLeft : Bool;   // Setup screen: executability of movement left
   //    movement3ExecutabilityRight : Bool;   // Setup screen: executability of movement right
   //    movement4ExecutabilityLeft : Bool;   // Setup screen: executability of movement left
   //    movement4ExecutabilityRight : Bool;   // Setup screen: executability of movement right
   //    movement5ExecutabilityLeft : Bool;   // Setup screen: executability of movement left
   //    movement5ExecutabilityRight : Bool;   // Setup screen: executability of movement right
   //    movement6ExecutabilityLeft : Bool;   // Setup screen: executability of movement left
   //    movement6ExecutabilityRight : Bool;   // Setup screen: executability of movement right
   //    movement7ExecutabilityLeft : Bool;   // Setup screen: executability of movement left
   //    movement7ExecutabilityRight : Bool;   // Setup screen: executability of movement right
   //    movement8ExecutabilityLeft : Bool;   // Setup screen: executability of movement left
   //    movement8ExecutabilityRight : Bool;   // Setup screen: executability of movement right
   //    movement9ExecutabilityLeft : Bool;   // Setup screen: executability of movement left
   //    movement9ExecutabilityRight : Bool;   // Setup screen: executability of movement right
   //    movement10ExecutabilityLeft : Bool;   // Setup screen: executability of movement left
   //    movement10ExecutabilityRight : Bool;   // Setup screen: executability of movement right
   //    movement11ExecutabilityLeft : Bool;   // Setup screen: executability of movement left
   //    movement11ExecutabilityRight : Bool;   // Setup screen: executability of movement right
   //    movement12ExecutabilityLeft : Bool;   // Setup screen: executability of movement left
   //    movement12ExecutabilityRight : Bool;   // Setup screen: executability of movement right
   //    movement13ExecutabilityLeft : Bool;   // Setup screen: executability of movement left
   //    movement13ExecutabilityRight : Bool;   // Setup screen: executability of movement right
   //    movement14ExecutabilityLeft : Bool;   // Setup screen: executability of movement left
   //    movement14ExecutabilityRight : Bool;   // Setup screen: executability of movement right
   //    movement15ExecutabilityLeft : Bool;   // Setup screen: executability of movement left
   //    movement15ExecutabilityRight : Bool;   // Setup screen: executability of movement right
   //    movement16ExecutabilityLeft : Bool;   // Setup screen: executability of movement left
   //    movement16ExecutabilityRight : Bool;   // Setup screen: executability of movement right
   //    movement17ExecutabilityLeft : Bool;   // Setup screen: executability of movement left
   //    movement17ExecutabilityRight : Bool;   // Setup screen: executability of movement right
   //    movement18ExecutabilityLeft : Bool;   // Setup screen: executability of movement left
   //    movement18ExecutabilityRight : Bool;   // Setup screen: executability of movement right
   //    movement19ExecutabilityLeft : Bool;   // Setup screen: executability of movement left
   //    movement19ExecutabilityRight : Bool;   // Setup screen: executability of movement right
   //    movement20ExecutabilityLeft : Bool;   // Setup screen: executability of movement left
   //    movement20ExecutabilityRight : Bool;   // Setup screen: executability of movement right
   //    movement21ExecutabilityLeft : Bool;   // Setup screen: executability of movement left
   //    movement21ExecutabilityRight : Bool;   // Setup screen: executability of movement right
   //    movement22ExecutabilityLeft : Bool;   // Setup screen: executability of movement left
   //    movement22ExecutabilityRight : Bool;   // Setup screen: executability of movement right
   //    movement23ExecutabilityLeft : Bool;   // Setup screen: executability of movement left
   //    movement23ExecutabilityRight : Bool;   // Setup screen: executability of movement right
   //    movement24ExecutabilityLeft : Bool;   // Setup screen: executability of movement left
   //    movement24ExecutabilityRight : Bool;   // Setup screen: executability of movement right
   //    movement25ExecutabilityLeft : Bool;   // Setup screen: executability of movement left
   //    movement25ExecutabilityRight : Bool;   // Setup screen: executability of movement right
   //    movement26ExecutabilityLeft : Bool;   // Setup screen: executability of movement left
   //    movement26ExecutabilityRight : Bool;   // Setup screen: executability of movement right
   //    movement27ExecutabilityLeft : Bool;   // Setup screen: executability of movement left
   //    movement27ExecutabilityRight : Bool;   // Setup screen: executability of movement right
   //    movement28ExecutabilityLeft : Bool;   // Setup screen: executability of movement left
   //    movement28ExecutabilityRight : Bool;   // Setup screen: executability of movement right
   //    movement29ExecutabilityLeft : Bool;   // Setup screen: executability of movement left
   //    movement29ExecutabilityRight : Bool;   // Setup screen: executability of movement right
   //    movement30ExecutabilityLeft : Bool;   // Setup screen: executability of movement left
   //    movement30ExecutabilityRight : Bool;   // Setup screen: executability of movement right
   //    movement31ExecutabilityLeft : Bool;   // Setup screen: executability of movement left
   //    movement31ExecutabilityRight : Bool;   // Setup screen: executability of movement right
   //    movement32ExecutabilityLeft : Bool;   // Setup screen: executability of movement left
   //    movement32ExecutabilityRight : Bool;   // Setup screen: executability of movement right
   //    movement33ExecutabilityLeft : Bool;   // Setup screen: executability of movement left
   //    movement33ExecutabilityRight : Bool;   // Setup screen: executability of movement right
   //    movement34ExecutabilityLeft : Bool;   // Setup screen: executability of movement left
   //    movement34ExecutabilityRight : Bool;   // Setup screen: executability of movement right
   //    movement35ExecutabilityLeft : Bool;   // Setup screen: executability of movement left
   //    movement35ExecutabilityRight : Bool;   // Setup screen: executability of movement right
   //    movement36ExecutabilityLeft : Bool;   // Setup screen: executability of movement left
   //    movement36ExecutabilityRight : Bool;   // Setup screen: executability of movement right
   //    movement37ExecutabilityLeft : Bool;   // Setup screen: executability of movement left
   //    movement37ExecutabilityRight : Bool;   // Setup screen: executability of movement right
   //    movement38ExecutabilityLeft : Bool;   // Setup screen: executability of movement left
   //    movement38ExecutabilityRight : Bool;   // Setup screen: executability of movement right
   //    movement39ExecutabilityLeft : Bool;   // Setup screen: executability of movement left
   //    movement39ExecutabilityRight : Bool;   // Setup screen: executability of movement right
   //    movement40ExecutabilityLeft : Bool;   // Setup screen: executability of movement left
   //    movement40ExecutabilityRight : Bool;   // Setup screen: executability of movement right
   //    movement41ExecutabilityLeft : Bool;   // Setup screen: executability of movement left
   //    movement41ExecutabilityRight : Bool;   // Setup screen: executability of movement right
   //    movement42ExecutabilityLeft : Bool;   // Setup screen: executability of movement left
   //    movement42ExecutabilityRight : Bool;   // Setup screen: executability of movement right
   //    movement43ExecutabilityLeft : Bool;   // Setup screen: executability of movement left
   //    movement43ExecutabilityRight : Bool;   // Setup screen: executability of movement right
   //    movement44ExecutabilityLeft : Bool;   // Setup screen: executability of movement left
   //    movement44ExecutabilityRight : Bool;   // Setup screen: executability of movement right
   //    movement45ExecutabilityLeft : Bool;   // Setup screen: executability of movement left
   //    movement45ExecutabilityRight : Bool;   // Setup screen: executability of movement right
   //    movement46ExecutabilityLeft : Bool;   // Setup screen: executability of movement left
   //    movement46ExecutabilityRight : Bool;   // Setup screen: executability of movement right
   //    movement47ExecutabilityLeft : Bool;   // Setup screen: executability of movement left
   //    movement47ExecutabilityRight : Bool;   // Setup screen: executability of movement right
   //    movement48ExecutabilityLeft : Bool;   // Setup screen: executability of movement left
   //    movement48ExecutabilityRight : Bool;   // Setup screen: executability of movement right
   //    movement49ExecutabilityLeft : Bool;   // Setup screen: executability of movement left
   //    movement49ExecutabilityRight : Bool;   // Setup screen: executability of movement right
   //    movement50ExecutabilityLeft : Bool;   // Setup screen: executability of movement left
   //    movement50ExecutabilityRight : Bool;   // Setup screen: executability of movement right
   //    movement51ExecutabilityLeft : Bool;   // Setup screen: executability of movement left
   //    movement51ExecutabilityRight : Bool;   // Setup screen: executability of movement right
   //    movement52ExecutabilityLeft : Bool;   // Setup screen: executability of movement left
   //    movement52ExecutabilityRight : Bool;   // Setup screen: executability of movement right
   //    movement53ExecutabilityLeft : Bool;   // Setup screen: executability of movement left
   //    movement53ExecutabilityRight : Bool;   // Setup screen: executability of movement right
   //    movement54ExecutabilityLeft : Bool;   // Setup screen: executability of movement left
   //    movement54ExecutabilityRight : Bool;   // Setup screen: executability of movement right
   //    movement55ExecutabilityLeft : Bool;   // Setup screen: executability of movement left
   //    movement55ExecutabilityRight : Bool;   // Setup screen: executability of movement right
   //    movement56ExecutabilityLeft : Bool;   // Setup screen: executability of movement left
   //    movement56ExecutabilityRight : Bool;   // Setup screen: executability of movement right
   //    movement57ExecutabilityLeft : Bool;   // Setup screen: executability of movement left
   //    movement57ExecutabilityRight : Bool;   // Setup screen: executability of movement right
   //    movement58ExecutabilityLeft : Bool;   // Setup screen: executability of movement left
   //    movement58ExecutabilityRight : Bool;   // Setup screen: executability of movement right
   //    movement59ExecutabilityLeft : Bool;   // Setup screen: executability of movement left
   //    movement59ExecutabilityRight : Bool;   // Setup screen: executability of movement right
   //    movement60ExecutabilityLeft : Bool;   // Setup screen: executability of movement left
   //    movement60ExecutabilityRight : Bool;   // Setup screen: executability of movement right
   //    movement61ExecutabilityLeft : Bool;   // Setup screen: executability of movement left
   //    movement61ExecutabilityRight : Bool;   // Setup screen: executability of movement right
   //    movement62ExecutabilityLeft : Bool;   // Setup screen: executability of movement left
   //    movement62ExecutabilityRight : Bool;   // Setup screen: executability of movement right
   //    movement63ExecutabilityLeft : Bool;   // Setup screen: executability of movement left
   //    movement63ExecutabilityRight : Bool;   // Setup screen: executability of movement right
   //    movement64ExecutabilityLeft : Bool;   // Setup screen: executability of movement left
   //    movement64ExecutabilityRight : Bool;   // Setup screen: executability of movement right
   //    movement65ExecutabilityLeft : Bool;   // Setup screen: executability of movement left
   //    movement65ExecutabilityRight : Bool;   // Setup screen: executability of movement right
   //    movement66ExecutabilityLeft : Bool;   // Setup screen: executability of movement left
   //    movement66ExecutabilityRight : Bool;   // Setup screen: executability of movement right
   //    movement67ExecutabilityLeft : Bool;   // Setup screen: executability of movement left
   //    movement67ExecutabilityRight : Bool;   // Setup screen: executability of movement right
   //    movement68ExecutabilityLeft : Bool;   // Setup screen: executability of movement left
   //    movement68ExecutabilityRight : Bool;   // Setup screen: executability of movement right
   //    movement69ExecutabilityLeft : Bool;   // Setup screen: executability of movement left
   //    movement69ExecutabilityRight : Bool;   // Setup screen: executability of movement right
   //    movement70ExecutabilityLeft : Bool;   // Setup screen: executability of movement left
   //    movement70ExecutabilityRight : Bool;   // Setup screen: executability of movement right
   //    movement71ExecutabilityLeft : Bool;   // Setup screen: executability of movement left
   //    movement71ExecutabilityRight : Bool;   // Setup screen: executability of movement right
   //    movement72ExecutabilityLeft : Bool;   // Setup screen: executability of movement left
   //    movement72ExecutabilityRight : Bool;   // Setup screen: executability of movement right
   //    movement73ExecutabilityLeft : Bool;   // Setup screen: executability of movement left
   //    movement73ExecutabilityRight : Bool;   // Setup screen: executability of movement right
   //    movement74ExecutabilityLeft : Bool;   // Setup screen: executability of movement left
   //    movement74ExecutabilityRight : Bool;   // Setup screen: executability of movement right
   //    movement75ExecutabilityLeft : Bool;   // Setup screen: executability of movement left
   //    movement75ExecutabilityRight : Bool;   // Setup screen: executability of movement right
   //    movement76ExecutabilityLeft : Bool;   // Setup screen: executability of movement left
   //    movement76ExecutabilityRight : Bool;   // Setup screen: executability of movement right
   //    movement77ExecutabilityLeft : Bool;   // Setup screen: executability of movement left
   //    movement77ExecutabilityRight : Bool;   // Setup screen: executability of movement right
   //    movement78ExecutabilityLeft : Bool;   // Setup screen: executability of movement left
   //    movement78ExecutabilityRight : Bool;   // Setup screen: executability of movement right
   //    movement79ExecutabilityLeft : Bool;   // Setup screen: executability of movement left
   //    movement79ExecutabilityRight : Bool;   // Setup screen: executability of movement right
   //    movement80ExecutabilityLeft : Bool;   // Setup screen: executability of movement left
   //    movement80ExecutabilityRight : Bool;   // Setup screen: executability of movement right
   //    movement81ExecutabilityLeft : Bool;   // Setup screen: executability of movement left
   //    movement81ExecutabilityRight : Bool;   // Setup screen: executability of movement right
   //    movement82ExecutabilityLeft : Bool;   // Setup screen: executability of movement left
   //    movement82ExecutabilityRight : Bool;   // Setup screen: executability of movement right
   //    movement83ExecutabilityLeft : Bool;   // Setup screen: executability of movement left
   //    movement83ExecutabilityRight : Bool;   // Setup screen: executability of movement right
   //    movement84ExecutabilityLeft : Bool;   // Setup screen: executability of movement left
   //    movement84ExecutabilityRight : Bool;   // Setup screen: executability of movement right
   //    movement85ExecutabilityLeft : Bool;   // Setup screen: executability of movement left
   //    movement85ExecutabilityRight : Bool;   // Setup screen: executability of movement right
   //    movement86ExecutabilityLeft : Bool;   // Setup screen: executability of movement left
   //    movement86ExecutabilityRight : Bool;   // Setup screen: executability of movement right
   //    movement87ExecutabilityLeft : Bool;   // Setup screen: executability of movement left
   //    movement87ExecutabilityRight : Bool;   // Setup screen: executability of movement right
   //    movement88ExecutabilityLeft : Bool;   // Setup screen: executability of movement left
   //    movement88ExecutabilityRight : Bool;   // Setup screen: executability of movement right
   //    movement89ExecutabilityLeft : Bool;   // Setup screen: executability of movement left
   //    movement89ExecutabilityRight : Bool;   // Setup screen: executability of movement right
   //    movement90ExecutabilityLeft : Bool;   // Setup screen: executability of movement left
   //    movement90ExecutabilityRight : Bool;   // Setup screen: executability of movement right
   //    movement91ExecutabilityLeft : Bool;   // Setup screen: executability of movement left
   //    movement91ExecutabilityRight : Bool;   // Setup screen: executability of movement right
   //    movement92ExecutabilityLeft : Bool;   // Setup screen: executability of movement left
   //    movement92ExecutabilityRight : Bool;   // Setup screen: executability of movement right
   //    movement93ExecutabilityLeft : Bool;   // Setup screen: executability of movement left
   //    movement93ExecutabilityRight : Bool;   // Setup screen: executability of movement right
   //    movement94ExecutabilityLeft : Bool;   // Setup screen: executability of movement left
   //    movement94ExecutabilityRight : Bool;   // Setup screen: executability of movement right
   //    movement95ExecutabilityLeft : Bool;   // Setup screen: executability of movement left
   //    movement95ExecutabilityRight : Bool;   // Setup screen: executability of movement right
   //    movement96ExecutabilityLeft : Bool;   // Setup screen: executability of movement left
   //    movement96ExecutabilityRight : Bool;   // Setup screen: executability of movement right
   //    movement97ExecutabilityLeft : Bool;   // Setup screen: executability of movement left
   //    movement97ExecutabilityRight : Bool;   // Setup screen: executability of movement right
   //    movement98ExecutabilityLeft : Bool;   // Setup screen: executability of movement left
   //    movement98ExecutabilityRight : Bool;   // Setup screen: executability of movement right
   //    movement99ExecutabilityLeft : Bool;   // Setup screen: executability of movement left
   //    movement99ExecutabilityRight : Bool;   // Setup screen: executability of movement right
   //    movement100ExecutabilityLeft : Bool;   // Setup screen: executability of movement left
   //    movement100ExecutabilityRight : Bool;   // Setup screen: executability of movement right
   //    movement101ExecutabilityLeft : Bool;   // Setup screen: executability of movement left
   //    movement101ExecutabilityRight : Bool;   // Setup screen: executability of movement right
   //    movement102ExecutabilityLeft : Bool;   // Setup screen: executability of movement left
   //    movement102ExecutabilityRight : Bool;   // Setup screen: executability of movement right
   //    movement103ExecutabilityLeft : Bool;   // Setup screen: executability of movement left
   //    movement103ExecutabilityRight : Bool;   // Setup screen: executability of movement right
   //    movement104ExecutabilityLeft : Bool;   // Setup screen: executability of movement left
   //    movement104ExecutabilityRight : Bool;   // Setup screen: executability of movement right
   //    movement105ExecutabilityLeft : Bool;   // Setup screen: executability of movement left
   //    movement105ExecutabilityRight : Bool;   // Setup screen: executability of movement right
   //    movement106ExecutabilityLeft : Bool;   // Setup screen: executability of movement left
   //    movement106ExecutabilityRight : Bool;   // Setup screen: executability of movement right
   //    movement107ExecutabilityLeft : Bool;   // Setup screen: executability of movement left
   //    movement107ExecutabilityRight : Bool;   // Setup screen: executability of movement right
   //    movement108ExecutabilityLeft : Bool;   // Setup screen: executability of movement left
   //    movement108ExecutabilityRight : Bool;   // Setup screen: executability of movement right
   //    movement109ExecutabilityLeft : Bool;   // Setup screen: executability of movement left
   //    movement109ExecutabilityRight : Bool;   // Setup screen: executability of movement right
   //    movement110ExecutabilityLeft : Bool;   // Setup screen: executability of movement left
   //    movement110ExecutabilityRight : Bool;   // Setup screen: executability of movement right
   //    movement111ExecutabilityLeft : Bool;   // Setup screen: executability of movement left
   //    movement111ExecutabilityRight : Bool;   // Setup screen: executability of movement right
   //    movement112ExecutabilityLeft : Bool;   // Setup screen: executability of movement left
   //    movement112ExecutabilityRight : Bool;   // Setup screen: executability of movement right
   //    movement113ExecutabilityLeft : Bool;   // Setup screen: executability of movement left
   //    movement113ExecutabilityRight : Bool;   // Setup screen: executability of movement right
   //    movement114ExecutabilityLeft : Bool;   // Setup screen: executability of movement left
   //    movement114ExecutabilityRight : Bool;   // Setup screen: executability of movement right
   //    movement115ExecutabilityLeft : Bool;   // Setup screen: executability of movement left
   //    movement115ExecutabilityRight : Bool;   // Setup screen: executability of movement right
   //    movement116ExecutabilityLeft : Bool;   // Setup screen: executability of movement left
   //    movement116ExecutabilityRight : Bool;   // Setup screen: executability of movement right
   //    movement117ExecutabilityLeft : Bool;   // Setup screen: executability of movement left
   //    movement117ExecutabilityRight : Bool;   // Setup screen: executability of movement right
   //    movement118ExecutabilityLeft : Bool;   // Setup screen: executability of movement left
   //    movement118ExecutabilityRight : Bool;   // Setup screen: executability of movement right
   //    movement119ExecutabilityLeft : Bool;   // Setup screen: executability of movement left
   //    movement119ExecutabilityRight : Bool;   // Setup screen: executability of movement right
   //    movement120ExecutabilityLeft : Bool;   // Setup screen: executability of movement left
   //    movement120ExecutabilityRight : Bool;   // Setup screen: executability of movement right
   //    movement121ExecutabilityLeft : Bool;   // Setup screen: executability of movement left
   //    movement121ExecutabilityRight : Bool;   // Setup screen: executability of movement right
   //    movement122ExecutabilityLeft : Bool;   // Setup screen: executability of movement left
   //    movement122ExecutabilityRight : Bool;   // Setup screen: executability of movement right
   //    movement123ExecutabilityLeft : Bool;   // Setup screen: executability of movement left
   //    movement123ExecutabilityRight : Bool;   // Setup screen: executability of movement right
   //    movement124ExecutabilityLeft : Bool;   // Setup screen: executability of movement left
   //    movement124ExecutabilityRight : Bool;   // Setup screen: executability of movement right
   //    movement125ExecutabilityLeft : Bool;   // Setup screen: executability of movement left
   //    movement125ExecutabilityRight : Bool;   // Setup screen: executability of movement right
   //    movement126ExecutabilityLeft : Bool;   // Setup screen: executability of movement left
   //    movement126ExecutabilityRight : Bool;   // Setup screen: executability of movement right
   //    movement127ExecutabilityLeft : Bool;   // Setup screen: executability of movement left
   //    movement127ExecutabilityRight : Bool;   // Setup screen: executability of movement right
   //    movement128ExecutabilityLeft : Bool;   // Setup screen: executability of movement left
   //    movement128ExecutabilityRight : Bool;   // Setup screen: executability of movement right
   //    movement129ExecutabilityLeft : Bool;   // Setup screen: executability of movement left
   //    movement129ExecutabilityRight : Bool;   // Setup screen: executability of movement right
   //    movement130ExecutabilityLeft : Bool;   // Setup screen: executability of movement left
   //    movement130ExecutabilityRight : Bool;   // Setup screen: executability of movement right
   //    movement131ExecutabilityLeft : Bool;   // Setup screen: executability of movement left
   //    movement131ExecutabilityRight : Bool;   // Setup screen: executability of movement right
   //    movement132ExecutabilityLeft : Bool;   // Setup screen: executability of movement left
   //    movement132ExecutabilityRight : Bool;   // Setup screen: executability of movement right
   //    movement133ExecutabilityLeft : Bool;   // Setup screen: executability of movement left
   //    movement133ExecutabilityRight : Bool;   // Setup screen: executability of movement right
   //    movement134ExecutabilityLeft : Bool;   // Setup screen: executability of movement left
   //    movement134ExecutabilityRight : Bool;   // Setup screen: executability of movement right
   //    movement135ExecutabilityLeft : Bool;   // Setup screen: executability of movement left
   //    movement135ExecutabilityRight : Bool;   // Setup screen: executability of movement right
   //    movement136ExecutabilityLeft : Bool;   // Setup screen: executability of movement left
   //    movement136ExecutabilityRight : Bool;   // Setup screen: executability of movement right
   //    movement137ExecutabilityLeft : Bool;   // Setup screen: executability of movement left
   //    movement137ExecutabilityRight : Bool;   // Setup screen: executability of movement right
   //    movement138ExecutabilityLeft : Bool;   // Setup screen: executability of movement left
   //    movement138ExecutabilityRight : Bool;   // Setup screen: executability of movement right
   //    movement139ExecutabilityLeft : Bool;   // Setup screen: executability of movement left
   //    movement139ExecutabilityRight : Bool;   // Setup screen: executability of movement right
   //    movement140ExecutabilityLeft : Bool;   // Setup screen: executability of movement left
   //    movement140ExecutabilityRight : Bool;   // Setup screen: executability of movement right
   //    movement141ExecutabilityLeft : Bool;   // Setup screen: executability of movement left
   //    movement141ExecutabilityRight : Bool;   // Setup screen: executability of movement right
   //    movement142ExecutabilityLeft : Bool;   // Setup screen: executability of movement left
   //    movement142ExecutabilityRight : Bool;   // Setup screen: executability of movement right
   //    movement143ExecutabilityLeft : Bool;   // Setup screen: executability of movement left
   //    movement143ExecutabilityRight : Bool;   // Setup screen: executability of movement right
   //    movement144ExecutabilityLeft : Bool;   // Setup screen: executability of movement left
   //    movement144ExecutabilityRight : Bool;   // Setup screen: executability of movement right
   //    movement145ExecutabilityLeft : Bool;   // Setup screen: executability of movement left
   //    movement145ExecutabilityRight : Bool;   // Setup screen: executability of movement right
   //    movement146ExecutabilityLeft : Bool;   // Setup screen: executability of movement left
   //    movement146ExecutabilityRight : Bool;   // Setup screen: executability of movement right
   //    movement147ExecutabilityLeft : Bool;   // Setup screen: executability of movement left
   //    movement147ExecutabilityRight : Bool;   // Setup screen: executability of movement right
   //    movement148ExecutabilityLeft : Bool;   // Setup screen: executability of movement left
   //    movement148ExecutabilityRight : Bool;   // Setup screen: executability of movement right
   //    movement149ExecutabilityLeft : Bool;   // Setup screen: executability of movement left
   //    movement149ExecutabilityRight : Bool;   // Setup screen: executability of movement right
   //    movement150ExecutabilityLeft : Bool;   // Setup screen: executability of movement left
   //    movement150ExecutabilityRight : Bool;   // Setup screen: executability of movement right
   //    movement151ExecutabilityLeft : Bool;   // Setup screen: executability of movement left
   //    movement151ExecutabilityRight : Bool;   // Setup screen: executability of movement right
   //    movement152ExecutabilityLeft : Bool;   // Setup screen: executability of movement left
   //    movement152ExecutabilityRight : Bool;   // Setup screen: executability of movement right
   //    movement153ExecutabilityLeft : Bool;   // Setup screen: executability of movement left
   //    movement153ExecutabilityRight : Bool;   // Setup screen: executability of movement right
   //    movement154ExecutabilityLeft : Bool;   // Setup screen: executability of movement left
   //    movement154ExecutabilityRight : Bool;   // Setup screen: executability of movement right
   //    movement155ExecutabilityLeft : Bool;   // Setup screen: executability of movement left
   //    movement155ExecutabilityRight : Bool;   // Setup screen: executability of movement right
   //    movement156ExecutabilityLeft : Bool;   // Setup screen: executability of movement left
   //    movement156ExecutabilityRight : Bool;   // Setup screen: executability of movement right
   //    movement157ExecutabilityLeft : Bool;   // Setup screen: executability of movement left
   //    movement157ExecutabilityRight : Bool;   // Setup screen: executability of movement right
   //    movement158ExecutabilityLeft : Bool;   // Setup screen: executability of movement left
   //    movement158ExecutabilityRight : Bool;   // Setup screen: executability of movement right
   //    movement159ExecutabilityLeft : Bool;   // Setup screen: executability of movement left
   //    movement159ExecutabilityRight : Bool;   // Setup screen: executability of movement right
   //    movement160ExecutabilityLeft : Bool;   // Setup screen: executability of movement left
   //    movement160ExecutabilityRight : Bool;   // Setup screen: executability of movement right
   //    movement161ExecutabilityLeft : Bool;   // Setup screen: executability of movement left
   //    movement161ExecutabilityRight : Bool;   // Setup screen: executability of movement right
   //    movement162ExecutabilityLeft : Bool;   // Setup screen: executability of movement left
   //    movement162ExecutabilityRight : Bool;   // Setup screen: executability of movement right
   //    movement163ExecutabilityLeft : Bool;   // Setup screen: executability of movement left
   //    movement163ExecutabilityRight : Bool;   // Setup screen: executability of movement right
   //    movement164ExecutabilityLeft : Bool;   // Setup screen: executability of movement left
   //    movement164ExecutabilityRight : Bool;   // Setup screen: executability of movement right
   //    movement165ExecutabilityLeft : Bool;   // Setup screen: executability of movement left
   //    movement165ExecutabilityRight : Bool;   // Setup screen: executability of movement right
   //    movement166ExecutabilityLeft : Bool;   // Setup screen: executability of movement left
   //    movement166ExecutabilityRight : Bool;   // Setup screen: executability of movement right
   //    movement167ExecutabilityLeft : Bool;   // Setup screen: executability of movement left
   //    movement167ExecutabilityRight : Bool;   // Setup screen: executability of movement right
   //    movement168ExecutabilityLeft : Bool;   // Setup screen: executability of movement left
   //    movement168ExecutabilityRight : Bool;   // Setup screen: executability of movement right
   //    movement169ExecutabilityLeft : Bool;   // Setup screen: executability of movement left
   //    movement169ExecutabilityRight : Bool;   // Setup screen: executability of movement right
   //    movement170ExecutabilityLeft : Bool;   // Setup screen: executability of movement left
   //    movement170ExecutabilityRight : Bool;   // Setup screen: executability of movement right
   //    movement171ExecutabilityLeft : Bool;   // Setup screen: executability of movement left
   //    movement171ExecutabilityRight : Bool;   // Setup screen: executability of movement right
   //    movement172ExecutabilityLeft : Bool;   // Setup screen: executability of movement left
   //    movement172ExecutabilityRight : Bool;   // Setup screen: executability of movement right
   //    movement173ExecutabilityLeft : Bool;   // Setup screen: executability of movement left
   //    movement173ExecutabilityRight : Bool;   // Setup screen: executability of movement right
   //    movement174ExecutabilityLeft : Bool;   // Setup screen: executability of movement left
   //    movement174ExecutabilityRight : Bool;   // Setup screen: executability of movement right
   //    movement175ExecutabilityLeft : Bool;   // Setup screen: executability of movement left
   //    movement175ExecutabilityRight : Bool;   // Setup screen: executability of movement right
   //    movement176ExecutabilityLeft : Bool;   // Setup screen: executability of movement left
   //    movement176ExecutabilityRight : Bool;   // Setup screen: executability of movement right
   //    movement177ExecutabilityLeft : Bool;   // Setup screen: executability of movement left
   //    movement177ExecutabilityRight : Bool;   // Setup screen: executability of movement right
   //    movement178ExecutabilityLeft : Bool;   // Setup screen: executability of movement left
   //    movement178ExecutabilityRight : Bool;   // Setup screen: executability of movement right
   //    movement179ExecutabilityLeft : Bool;   // Setup screen: executability of movement left
   //    movement179ExecutabilityRight : Bool;   // Setup screen: executability of movement right
   //    movement180ExecutabilityLeft : Bool;   // Setup screen: executability of movement left
   //    movement180ExecutabilityRight : Bool;   // Setup screen: executability of movement right
   //    movement181ExecutabilityLeft : Bool;   // Setup screen: executability of movement left
   //    movement181ExecutabilityRight : Bool;   // Setup screen: executability of movement right
   //    movement182ExecutabilityLeft : Bool;   // Setup screen: executability of movement left
   //    movement182ExecutabilityRight : Bool;   // Setup screen: executability of movement right
   //    movement183ExecutabilityLeft : Bool;   // Setup screen: executability of movement left
   //    movement183ExecutabilityRight : Bool;   // Setup screen: executability of movement right
   //    movement184ExecutabilityLeft : Bool;   // Setup screen: executability of movement left
   //    movement184ExecutabilityRight : Bool;   // Setup screen: executability of movement right
   //    movement185ExecutabilityLeft : Bool;   // Setup screen: executability of movement left
   //    movement185ExecutabilityRight : Bool;   // Setup screen: executability of movement right
   //    movement186ExecutabilityLeft : Bool;   // Setup screen: executability of movement left
   //    movement186ExecutabilityRight : Bool;   // Setup screen: executability of movement right
   //    movement187ExecutabilityLeft : Bool;   // Setup screen: executability of movement left
   //    movement187ExecutabilityRight : Bool;   // Setup screen: executability of movement right
   //    movement188ExecutabilityLeft : Bool;   // Setup screen: executability of movement left
   //    movement188ExecutabilityRight : Bool;   // Setup screen: executability of movement right
   //    movement189ExecutabilityLeft : Bool;   // Setup screen: executability of movement left
   //    movement189ExecutabilityRight : Bool;   // Setup screen: executability of movement right
   //    movement190ExecutabilityLeft : Bool;   // Setup screen: executability of movement left
   //    movement190ExecutabilityRight : Bool;   // Setup screen: executability of movement right
   //    movement191ExecutabilityLeft : Bool;   // Setup screen: executability of movement left
   //    movement191ExecutabilityRight : Bool;   // Setup screen: executability of movement right
   //    movement192ExecutabilityLeft : Bool;   // Setup screen: executability of movement left
   //    movement192ExecutabilityRight : Bool;   // Setup screen: executability of movement right
   //    movement193ExecutabilityLeft : Bool;   // Setup screen: executability of movement left
   //    movement193ExecutabilityRight : Bool;   // Setup screen: executability of movement right
   //    movement194ExecutabilityLeft : Bool;   // Setup screen: executability of movement left
   //    movement194ExecutabilityRight : Bool;   // Setup screen: executability of movement right
   //    movement195ExecutabilityLeft : Bool;   // Setup screen: executability of movement left
   //    movement195ExecutabilityRight : Bool;   // Setup screen: executability of movement right
   //    movement196ExecutabilityLeft : Bool;   // Setup screen: executability of movement left
   //    movement196ExecutabilityRight : Bool;   // Setup screen: executability of movement right
   //    movement197ExecutabilityLeft : Bool;   // Setup screen: executability of movement left
   //    movement197ExecutabilityRight : Bool;   // Setup screen: executability of movement right
   //    movement198ExecutabilityLeft : Bool;   // Setup screen: executability of movement left
   //    movement198ExecutabilityRight : Bool;   // Setup screen: executability of movement right
   //    movement199ExecutabilityLeft : Bool;   // Setup screen: executability of movement left
   //    movement199ExecutabilityRight : Bool;   // Setup screen: executability of movement right
   //    movement200ExecutabilityLeft : Bool;   // Setup screen: executability of movement left
   //    movement200ExecutabilityRight : Bool;   // Setup screen: executability of movement right
   //    movement201ExecutabilityLeft : Bool;   // Setup screen: executability of movement left
   //    movement201ExecutabilityRight : Bool;   // Setup screen: executability of movement right
   //    movement202ExecutabilityLeft : Bool;   // Setup screen: executability of movement left
   //    movement202ExecutabilityRight : Bool;   // Setup screen: executability of movement right
   //    movement203ExecutabilityLeft : Bool;   // Setup screen: executability of movement left
   //    movement203ExecutabilityRight : Bool;   // Setup screen: executability of movement right
   //    movement204ExecutabilityLeft : Bool;   // Setup screen: executability of movement left
   //    movement204ExecutabilityRight : Bool;   // Setup screen: executability of movement right
   //    movement205ExecutabilityLeft : Bool;   // Setup screen: executability of movement left
   //    movement205ExecutabilityRight : Bool;   // Setup screen: executability of movement right
   //    movement206ExecutabilityLeft : Bool;   // Setup screen: executability of movement left
   //    movement206ExecutabilityRight : Bool;   // Setup screen: executability of movement right
   //    movement207ExecutabilityLeft : Bool;   // Setup screen: executability of movement left
   //    movement207ExecutabilityRight : Bool;   // Setup screen: executability of movement right
   //    movement208ExecutabilityLeft : Bool;   // Setup screen: executability of movement left
   //    movement208ExecutabilityRight : Bool;   // Setup screen: executability of movement right
   //    movement209ExecutabilityLeft : Bool;   // Setup screen: executability of movement left
   //    movement209ExecutabilityRight : Bool;   // Setup screen: executability of movement right
   //    movement210ExecutabilityLeft : Bool;   // Setup screen: executability of movement left
   //    movement210ExecutabilityRight : Bool;   // Setup screen: executability of movement right
   //    movement211ExecutabilityLeft : Bool;   // Setup screen: executability of movement left
   //    movement211ExecutabilityRight : Bool;   // Setup screen: executability of movement right
   //    movement212ExecutabilityLeft : Bool;   // Setup screen: executability of movement left
   //    movement212ExecutabilityRight : Bool;   // Setup screen: executability of movement right
   //    movement213ExecutabilityLeft : Bool;   // Setup screen: executability of movement left
   //    movement213ExecutabilityRight : Bool;   // Setup screen: executability of movement right
   //    movement214ExecutabilityLeft : Bool;   // Setup screen: executability of movement left
   //    movement214ExecutabilityRight : Bool;   // Setup screen: executability of movement right
   //    movement215ExecutabilityLeft : Bool;   // Setup screen: executability of movement left
   //    movement215ExecutabilityRight : Bool;   // Setup screen: executability of movement right
   //    movement216ExecutabilityLeft : Bool;   // Setup screen: executability of movement left
   //    movement216ExecutabilityRight : Bool;   // Setup screen: executability of movement right
   //    movement217ExecutabilityLeft : Bool;   // Setup screen: executability of movement left
   //    movement217ExecutabilityRight : Bool;   // Setup screen: executability of movement right
   //    movement218ExecutabilityLeft : Bool;   // Setup screen: executability of movement left
   //    movement218ExecutabilityRight : Bool;   // Setup screen: executability of movement right
   //    movement219ExecutabilityLeft : Bool;   // Setup screen: executability of movement left
   //    movement219ExecutabilityRight : Bool;   // Setup screen: executability of movement right
   //    movement220ExecutabilityLeft : Bool;   // Setup screen: executability of movement left
   //    movement220ExecutabilityRight : Bool;   // Setup screen: executability of movement right
   //    movement221ExecutabilityLeft : Bool;   // Setup screen: executability of movement left
   //    movement221ExecutabilityRight : Bool;   // Setup screen: executability of movement right
   //    movement222ExecutabilityLeft : Bool;   // Setup screen: executability of movement left
   //    movement222ExecutabilityRight : Bool;   // Setup screen: executability of movement right
   //    movement223ExecutabilityLeft : Bool;   // Setup screen: executability of movement left
   //    movement223ExecutabilityRight : Bool;   // Setup screen: executability of movement right
   //    movement224ExecutabilityLeft : Bool;   // Setup screen: executability of movement left
   //    movement224ExecutabilityRight : Bool;   // Setup screen: executability of movement right
   //    movement225ExecutabilityLeft : Bool;   // Setup screen: executability of movement left
   //    movement225ExecutabilityRight : Bool;   // Setup screen: executability of movement right
   //    movement226ExecutabilityLeft : Bool;   // Setup screen: executability of movement left
   //    movement226ExecutabilityRight : Bool;   // Setup screen: executability of movement right
   //    movement227ExecutabilityLeft : Bool;   // Setup screen: executability of movement left
